PROGRAM MAIN
VAR
END_VAR

IF _TaskInfo[GETCURTASKINDEXEX()].FirstCycle THEN
	F_Log(E_LogLevel.eInfo, 'SPS Task gestartet.');
END_IF

PRG_TaskLog.Call();

END_PROGRAM

(* stored: Version 1.1.0.1, ProductVersion 3.1.4024.0
   POU MAIN: Id {0d65efd7-894c-4144-a23c-4d79bdbdc725}, SpecialFunc None *)
